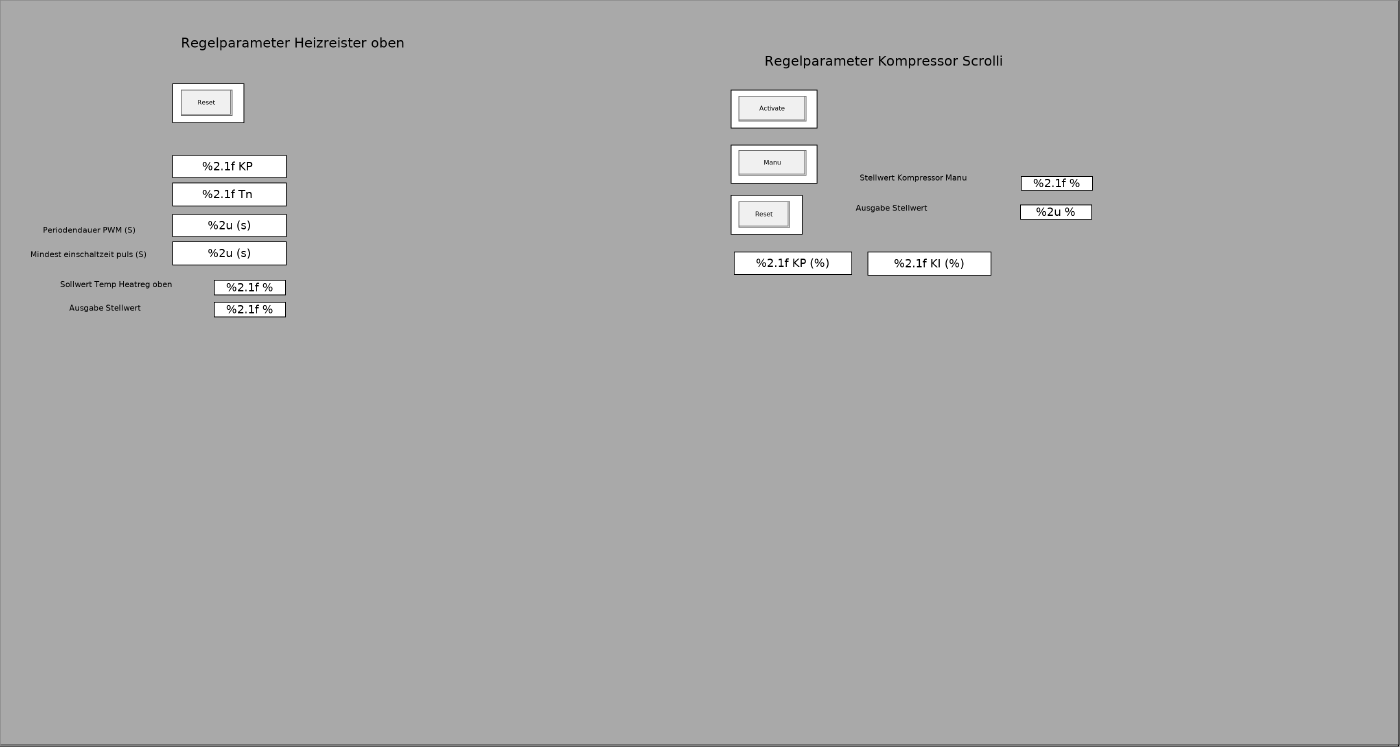
VISUALIZATION Service  // 1780x950
    Rectangle (203,38 339x33), "Regelparameter Heizreister oben"
    Rectangle (272,384 91x19), "%2.1f %", tooltip "Durchmesser in mm eingeben", text variable: fTemp_mean_belt_top
    Rectangle (44,383 179x17), "Ausgabe Stellwert"
    Rectangle (219,106 91x50)
    Button (230,114 65x33), "Reset"
        tap Reset_heatreg_top
    Rectangle (219,197 145x29), "%2.1f KP", tooltip "Durchmesser in mm eingeben", text variable: fKP_Controller_Heatmatt1
        OnMouseDown: write the text variable via VisuDialogs.Numpad, min 0, max 100
    Rectangle (219,232 145x30), "%2.1f Tn", tooltip "Durchmesser in mm eingeben", text variable: fKI_Controller_Heatmatt1
        OnMouseDown: write the text variable via VisuDialogs.Numpad, min 0, max 100
    Rectangle (272,356 91x19), "%2.1f %", tooltip "Durchmesser in mm eingeben", text variable: fSetpointValue1
        OnMouseDown: write the text variable via VisuDialogs.Numpad, min 0, max 100
    Rectangle (29,345 238x33), "Sollwert Temp Heatreg oben"
    Group (919,61 470x289)
        Rectangle (0,0 409x33), "Regelparameter Kompressor Scrolli"
        Rectangle (379,163 91x18), "%2.1f %", tooltip "Durchmesser in mm eingeben", text variable: GVL.fManual_controller_comp
            OnMouseDown: write the text variable via VisuDialogs.Numpad, min 0, max 100
        Rectangle (10,123 110x49), colour toggle: GVL.Set_Manual_controller_comp
        Button (20,130 86x32), "Manu", pressed state: GVL.Set_Manual_controller_comp
            toggle GVL.Set_Manual_controller_comp
        Rectangle (378,199 91x19), "%2u %", tooltip "Durchmesser in mm eingeben", text variable: GVL.fStellwert_comp
        Rectangle (125,195 179x17), "Ausgabe Stellwert"
        Rectangle (10,187 91x50), colour toggle: GVL.Reset_Controller_comp
        Button (20,195 65x33), "Reset"
            tap GVL.Reset_Controller_comp
        Rectangle (14,259 150x29), "%2.1f KP (%)", tooltip "Durchmesser in mm eingeben", text variable: GVL.fKP_Controller_comp
            OnMouseDown: write the text variable via VisuDialogs.Numpad, min 0, max 100
        Rectangle (184,259 157x30), "%2.1f KI (%)", tooltip "Durchmesser in mm eingeben", text variable: GVL.fKI_Controller_comp
            OnMouseDown: write the text variable via VisuDialogs.Numpad, min 0, max 100
        Rectangle (131,156 223x18), "Stellwert Kompressor Manu"
        Rectangle (10,53 110x49), colour toggle: GVL.Activate_controller_comp
        Button (20,61 86x32), "Activate", pressed state: GVL.Activate_controller_comp
            toggle GVL.Activate_controller_comp
    Rectangle (1778,0 2x947)
    Rectangle (0,947 1778x3)
    Rectangle (219,272 145x29), "%2u (s)", tooltip "Durchmesser in mm eingeben", text variable: udiPrd_heatreg1
        OnMouseDown: write the text variable via VisuDialogs.Numpad, min 0, max 100
    Rectangle (219,307 145x30), "%2u (s)", tooltip "Durchmesser in mm eingeben", text variable: udiMinOnTi_heatreg_1
        OnMouseDown: write the text variable via VisuDialogs.Numpad, min 0, max 100
    Rectangle (24,284 179x17), "Periodendauer PWM (S)"
    Rectangle (23,315 179x17), "Mindest einschaltzeit puls (S)"
END_VISUALIZATION

(* stored: Version 1.1.0.1, ProductVersion 3.1.4024.3
   Visu Service: Id {b729f37b-ef59-4469-ba27-acae8e633791} *)
